PROGRAM MAIN2
VAR	

	// ========= System Control / FSM Variables =========
	
	MainCommands 		: MainCommands_typ; 		// command struct for cycling thru the state machine
	MainState    		: MainStateMachine_enum;   	// enumeration for the Main state machine
	System				: Mediator;					// System-level control object

	// ========= Linked NC Variables & References =========
	
	Mover    			: ARRAY[0..GVL.NUM_MOVERS - 1] OF Mover; 	// instantiation of Mover objects. Matches the number of movers on the system
	
	// ========= Objectives & Parameters =========

	ParameterSet		: MotionParameters_typ;
	
	MoverList			: ARRAY[0..GVL.NUM_MOVERLISTS-1] OF MoverList;
	PositionTrigger		: ARRAY[0..GVL.NUM_POSITIONTRIGGERS-1] OF PositionTrigger;
	Station				: ARRAY[0..GVL.NUM_STATIONS-1] OF Station;
	Track				: ARRAY[0..GVL.NUM_TRACKS] OF Track;
	Zone				: ARRAY[0..GVL.NUM_ZONES-1] OF Zone;
	
    // ========= Helper, State, & Index Variables =========
	
    i                	: UINT; 	// index variable; gets reused in various FOR loops
    n                	: UINT; 	// secondary index variable, for enabling movers
	
	// ========= XTS Utility Diagnostics =========
	
	nEnvironmentState				: INT;
	
	// ========= Example Application Variables =========

    nextStation 		: USINT := 4;
                    	
    lowVelocity    		: LREAL := 200;  	// mm/s
    mediumVelocity 		: LREAL := 800;  	// mm/s
    highVelocity   		: LREAL := 1200; 	// mm/s
	
	StationTimer 		: ARRAY[0..GVL.NUM_STATIONS] OF TON; // timer blocks, for station dwells
END_VAR

EnvironmentCyclic();

CASE MainState OF
	MainStateMachine_enum.MS_DISABLED: // ------------------------------------------
	
		// XTS is idle. Motive power is disabled.	
		IF MainCommands.Enable THEN
			MainCommands.Disable			:= FALSE;
			MainCommands.Stop				:= FALSE;
			MainState						:= MainStateMachine_enum.MS_INITIALIZING;
		END_IF

	MainStateMachine_enum.MS_INITIALIZING: // --------------------------------------
	
		Registering();			// Add all objectives & movers to the system-level Mediator object
		Initializing();			// Set basic application parameters for the objects
			
		System.CompleteMoverList.EnableAll();
		System.CompleteMoverList.ActivateAllTrack( Track[1] );
		
		IF System.CompleteMoverList.IsAllTrackReady AND System.CompleteMoverList.IsAllMoversReady THEN
			MainState	:= MainStateMachine_enum.MS_ENABLED;
		END_IF
	
	MainStateMachine_enum.MS_ENABLED:	// -------------------------------------------
	
		// Recovery logic
		IF MainCommands.Start THEN
			System.CompleteMoverList.MoveAllToStation( Station[0] );
			System.ResetStatistics();
			// Reinit nextStation
        	nextStation := 4;
			MainState			:= MainStateMachine_enum.MS_RUN;
		ELSIF MainCommands.Disable THEN
			MainCommands.Enable	:= FALSE;
			System.CompleteMoverList.HaltAll();
			MainState			:= MainStateMachine_enum.MS_STOPPING;
			
		END_IF
	
	MainStateMachine_enum.MS_RUN: // -----------------------------------------------
	
		StationLogic();
	
        IF MainCommands.Stop THEN
            MainCommands.Start 	:= FALSE;
			System.CompleteMoverList.HaltAll();
            MainState         	:= MainStateMachine_enum.MS_STOPPING;
        ELSIF MainCommands.Disable THEN
            MainCommands.Enable := FALSE;
			System.CompleteMoverList.HaltAll();
            MainState           := MainStateMachine_enum.MS_STOPPING;
        END_IF
		
	MainStateMachine_enum.MS_STOPPING:
	
		IF System.CompleteMoverList.IsAllMoversHalted THEN
			MainState			:= MainStateMachine_enum.MS_STOPPED;
		END_IF
		
	MainStateMachine_enum.MS_STOPPED: // -------------------------------------------
	
	    IF MainCommands.Disable THEN
            MainCommands.Enable 	:= FALSE;
			MainCommands.Start		:= FALSE;
			System.CompleteMoverList.DisableAll();
            MainState           	:= MainStateMachine_enum.MS_DISABLING;
        ELSIF MainCommands.Start THEN
            MainCommands.Stop 		:= FALSE;
            MainState         		:= MainStateMachine_enum.MS_ENABLED;
        END_IF
		
	MainStateMachine_enum.MS_DISABLING: // -------------------------------------------
	
		IF System.CompleteMoverList.IsAllMoversDisabled THEN
			MainState			:= MainStateMachine_enum.MS_DISABLED;
		END_IF
		
	MainStateMachine_enum.MS_ERROR: // ---------------------------------------------
	MainStateMachine_enum.MS_DEBUG: // ---------------------------------------------	
	

END_CASE

System.Cyclic();

ACTION EnvironmentCyclic:
CASE nEnvironmentState OF
	0:	// ----------------------------------------- Enable Init Items
	
		// Enable init Info Server if needed
		ENV.stXtsEnvironmentConfiguration.bEnableInitInfoServer		:= TRUE;
		
		// Enable init CA Group if needed
		ENV.stXtsEnvironmentConfiguration.bEnableInitCaGroup		:= TRUE;
		
		// Set configuration of XtsUtility init
		ENV.fbXtsEnvironment.P_XtsEnvironmentConfiguration			:= ENV.stXtsEnvironmentConfiguration;
		
		// Next step
		nEnvironmentState	:= 1;
		
	1:	// ------------------------------------------ Init Environment
		
		// Start init
		IF ENV.fbXtsEnvironment.Init(TRUE) THEN
			// stop init
			ENV.fbXtsEnvironment.Init(FALSE);
			
			// next step
			nEnvironmentState	:= 2;
		END_IF
		
	2:	// ------------------------------------------ Check for success
	
		// Check IsInitialized property
		IF ENV.fbXtsEnvironment.P_IsInitialized THEN
			// next step
			nEnvironmentState	:= 3;
		END_IF
		
	3:	// ------------------------------------------- Init Visu
	
		ENV.fbXtsEnvironmentVisu( ipTcIoXtsEnvironment := ENV.fbXtsEnvironment );
		
		// next step
		nEnvironmentState	:= 4;
		
	4:	// ------------------------------------------- Init done

		ENV.fbXtsEnvironmentVisu.Cycle();
		
END_CASE
END_ACTION

ACTION Initializing:


	// Initialize station positions
	Station[0].Position 		:= 5;
	Station[1].Position 		:= 750;
	Station[2].Position 		:= 1200;
	Station[3].Position 		:= 1300;
	Station[4].Position 		:= 1400;

	PositionTrigger[0].Position := 1500;
	PositionTrigger[1].Position := 2000;
	PositionTrigger[2].Position := 3500;

	Zone[0].StartPosition		:= 3750;
	Zone[0].EndPosition   		:= 750;

	Zone[1].StartPosition 		:= 750;
	Zone[1].EndPosition   		:= 1750;

	Zone[2].StartPosition 		:= 1750;
	Zone[2].EndPosition   		:= 2750;

	Zone[3].StartPosition		:= 2750;
	Zone[3].EndPosition   		:= 3750;
	
	System.CompleteMoverList.SetAllVelocity( 1E3 );
	System.CompleteMoverList.SetAllAcceleration( 1E4 );
	System.CompleteMoverList.SetAllDeceleration( 1E4 );
	System.CompleteMoverList.SetAllJerk( 5E5 );
	System.CompleteMoverList.SetAllGap( 85 );
	System.CompleteMoverList.SetAllDirection( mcDirectionPositive );
END_ACTION

ACTION Registering:
	

		// Add all Movers to the Mediator
		FOR i := 0 TO GVL.NUM_MOVERS - 1 DO
			System.AddMover( Mover[i] );
		END_FOR
	
		// Add all Mover Lists to the Mediator
		FOR i := 0 TO GVL.NUM_MOVERLISTS - 1 DO
			System.AddMoverList( MoverList[i] );
		END_FOR
		
		// Add all PositionTriggers to the Mediator
		FOR i := 0 TO GVL.NUM_POSITIONTRIGGERS - 1 DO
			System.AddPositionTrigger( PositionTrigger[i] );
		END_FOR
		
		// Add all Stations to the Mediator
		FOR i := 0 TO GVL.NUM_STATIONS - 1 DO
			System.AddStation( Station[i] );
		END_FOR
		
		// Add all Tracks to the Mediator
		// note track zero is a special case, so the loop is one larger than the rest of the initalization loops
		FOR i := 0 TO GVL.NUM_TRACKS DO
			Track[i].Id := UINT_TO_INT(i);
			System.AddTrack( Track[i] );
		END_FOR
		
		// Add all Zones to the Mediator
		FOR i := 0 TO GVL.NUM_ZONES - 1 DO
			System.AddZone( Zone[i] );
		END_FOR
END_ACTION

ACTION StationLogic:
		(*Mover routing logic should be written here to define the system's operating behavior.
		Station implementations, Position Trigger logic, etc. In general, you can remove the example code
		here down to the short line break that looks like this: // ============= *)
	
        // Station 0 Logic
        IF Station[0].MoverInPosition THEN
            StationTimer[0](IN := TRUE, PT := T#1000MS);
            IF StationTimer[0].Q THEN
                Station[0].CurrentMover.SetVelocity(mediumVelocity);
                Station[0].CurrentMover.MoveToStation(Station[1]);
            END_IF
        ELSE
            StationTimer[0](IN := FALSE);
        END_IF
		
        // Station 1 Logic		
        IF Station[1].MoverInPosition THEN
            StationTimer[1](IN := TRUE, PT := T#250MS);
            IF StationTimer[1].Q THEN
                Station[1].CurrentMover.SetVelocity(mediumVelocity);
                Station[1].CurrentMover.MoveToStation(Station[nextStation]);
                nextStation := nextStation - 1;
                IF nextStation = 1 THEN
                    nextStation := 4;
                END_IF
            END_IF
        ELSE
            StationTimer[1](IN := FALSE);
        END_IF
		
		// Group of Stations 2, 3, and 4 Logic
        IF Station[2].MoverInPosition AND Station[3].MoverInPosition AND Station[4].MoverInPosition THEN
            StationTimer[2](IN := TRUE, PT := T#750MS);
            IF StationTimer[2].Q THEN
				StationTimer[2](IN := FALSE);

                Station[2].CurrentMover.MoveVelocity(500);
                Station[3].CurrentMover.MoveVelocity(500);
                Station[4].CurrentMover.MoveVelocity(500);
            END_IF
        END_IF
		
        // Position Trigger 0 Logic
        IF PositionTrigger[0].MoverPassedPosition THEN
            PositionTrigger[0].CurrentMover.SetVelocity(lowVelocity);
            PositionTrigger[0].MuteCurrent();
        END_IF
		
        // Position Trigger 1 Logic
        IF PositionTrigger[1].MoverPassedPosition THEN
            PositionTrigger[1].CurrentMover.SetVelocity(highVelocity);
            PositionTrigger[1].MuteCurrent();
        END_IF

		// Position Trigger 2 Logic
        IF PositionTrigger[2].MoverPassedPosition THEN
            PositionTrigger[2].CurrentMover.SetVelocity(lowVelocity);
            PositionTrigger[2].CurrentMover.MoveToStation(Station[0]);
            PositionTrigger[2].MuteCurrent();
        END_IF
END_ACTION

END_PROGRAM

(* stored: Version 1.1.0.1, ProductVersion 3.1.4024.12
   POU MAIN2: Id {c992ed33-41fe-02c4-17ef-23123b9a5b23}, SpecialFunc None
   Action EnvironmentCyclic: Id {9a903fbd-e9ae-032f-2559-00badaf47834}
   Action Initializing: Id {77eee1d6-568e-0448-2c64-a85af70fbf71}
   Action Registering: Id {ef3ef836-2b88-0099-2899-1cd10004220b}
   Action StationLogic: Id {ad15b1d3-f9a4-013e-29dd-5430b02980cb} *)
